FUNCTION_BLOCK FB_EstacionFinalizar_SFC
VAR_INPUT
    // SFC-Flags
    SFCPause: BOOL;
    SFCReset: BOOL;
    
    // Indicadores de sincronizacion
    Benido: BOOL := TRUE;
    Ejecuta: BOOL;
    
    // Parametros
    TpoFinalizacion: TIME := T#1S;
END_VAR
VAR_OUTPUT
    // Indicadores de sincronizacion
    Acabhe: BOOL;
    ListoKalisto: BOOL;
END_VAR
VAR
END_VAR

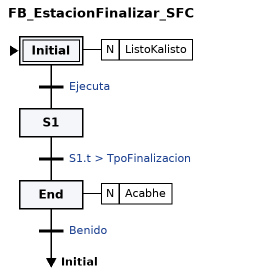
INITIAL_STEP Initial:
    ListoKalisto(N);
END_STEP
TRANSITION FROM Initial TO S1
    := Ejecuta;
END_TRANSITION
STEP S1:
END_STEP
TRANSITION FROM S1 TO End
    := S1.t > TpoFinalizacion;
END_TRANSITION
STEP End:
    Acabhe(N);
END_STEP
TRANSITION FROM End TO Initial
    := Benido;
END_TRANSITION

END_FUNCTION_BLOCK

(* stored: Version 1.1.0.1, ProductVersion 3.1.4024.12
   POU FB_EstacionFinalizar_SFC: Id {5150e515-81ce-47a4-a5df-bc4e8651597a}, SpecialFunc None *)
